TYPE stMotorCtrl :
STRUCT
	rTpoAcelDecel :REAL; // Tiempo para acelerar/decelerar hasta alcanazar la velocidad.
	rVelRpm       :REAL; // Velocidad en RPM.
	xMotorOff     :BOOL; // Bit de paro ON.
	xMotorOn      :BOOL   ; // Bit de marcha OFF.	
END_STRUCT
END_TYPE

(* stored: Version 1.1.0.1, ProductVersion 3.1.4024.12
   DUT stMotorCtrl: Id {2fa7d62e-97b0-453c-a8f1-3cee677f3d5f} *)
